(* This Program Show The Timer Patter Used for PLC *)

PROGRAM main
VAR
	TON0 : TON;
	Timer : time := T#5s;
	Time_Counter : time;
	Start : bool;
	Output : bool;
END_VAR

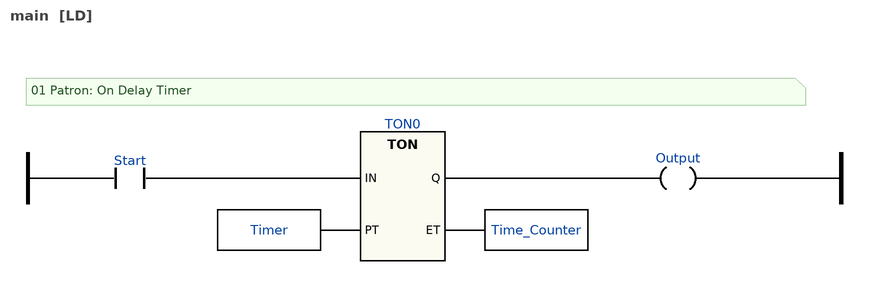
(* LD diagram, written out as Structured Text *)
(* 01 Patron: On Delay Timer *)
TON0(IN := Start, PT := Timer);
Output := TON0.Q;
Time_Counter := TON0.ET;
END_PROGRAM
